FUNCTION FC_Pt100Raw_TO_Temperature : REAL
VAR_INPUT
	i : REAL;
END_VAR
VAR
	ConvFac : REAL := 10;
END_VAR

FC_Pt100Raw_TO_Temperature := (i)/ConvFac;

END_FUNCTION

(* stored: Version 1.1.0.1, ProductVersion 3.1.4024.3
   POU FC_Pt100Raw_TO_Temperature: Id {6cfe8a6d-d01e-4d22-bc2b-00d23a3d6bc3}, SpecialFunc None *)
